Staubli VAL3: io_System.dtx

public num nLiAuto
public num nLiAux1
public num nLiAux2
public num nLiAux3
public num nLiDoorOpen
public num nLiEnd
public num nLiHome = 1
public num nLiMouldFree
public num nLiPartMade
public num nLiRobotOff
public num nLiSafety
public num nLiStart
public num nLiStop = 1
public num nLiTotalHome = 1
public num nLiWarning
public num nStateRobot
public num nLiTowerRed
public num nLiTowerYellow
public num nLiTowerGreen
public num nPowerCountCtrl
public num nLastServiceCtr
public num nLastServiceArm
public num nServiceRemain
public string sAux1
public string sAux2
public bool bBlockedCycle
public bool bBlockedUser
public bool bBtEnd
public bool bBtHome
public bool bBtRobotOff
public bool bBtStart
public bool bBtStop
public bool bCancelHomeCycl
public bool bCycleEndCalled
public bool bCycleEndPos
public bool bEnd
public bool bF7
public bool bF8
public bool bF_End
public bool bF_Home
public bool bF_Off
public bool bF_Start
public bool bF_Stop
public bool bFirstRunAfterL = true
public bool bFlashFast
public bool bFlashSlow
public bool bForceHomeReq
public bool bForceHome_ = true
public bool bHomeRetActive
public bool bModified
public bool bMouldArmInPLC
public bool bPartMade
public bool bRobotHome = true
public bool bRobotOff
public bool bRobotOffCalled
public bool bRobotOffPos
public bool bRobotZero
public bool bStartHomeCycle
public bool bStartProdCycle
public bool bTotalHome = true
public bool bUsrError
public bool btAux1
public bool btAux2
public bool btAux3
public bool bUsrWarningLow
public bool canStart
public bool canStop
public bool canResume
public bool canHom
public bool canRobotOff
public bool bRecordForce
public bool bErrorAck
public bool bUsrWarningHigh
public bool bIsEmulator
public bool bCancelEndCycle
public bool bStartInEndCycl
public jointRx jEnvMax = {j1=88.269052, j2=85.051261, j3=143.532119, j4=182.33531, j5=117.927529, j6=254.739889}
public jointRx jEnvMin = {j1=-180, j2=-47.382245, j3=-142.046726, j4=-131.97883, j5=-69.877872, j6=-189.153148}
public jointRx jPosErrCurrent = {j1=5.7E-05, j4=6.1E-05}
public jointRx jTorqueCurrent
public aio aiGrip[9]
public dio diArm[9]
public dio diBtAux1
public dio diBtAux2
public dio diBtAux3
public dio diBtEnd
public dio diBtHome
public dio diBtRobotOff
public dio diBtStart
public dio diBtStop
public dio diBtTotalHome
public dio diCore1Pos1
public dio diCore1Pos2
public dio diCore2Pos1
public dio diCore2Pos2
public dio diEjcIn
public dio diEjcOut
public dio diGrip[9]
public dio diGrip2[9]
public dio diLifeBit[2]
public dio diMachineInAuto
public dio diMouldClosed
public dio diMouldFreeFBK
public dio diMouldMidOpen
public dio diMouldOpen
public dio diRejectPart
public dio diSecuFBK[2]
public dio doAir[9]
public dio doArm[9]
public dio doAux1
public dio doAux2
public dio doCore1Pos1
public dio doCore1Pos2
public dio doCore2Pos1
public dio doCore2Pos2
public dio doEjcIn
public dio doEjcOut
public dio doFullOpening
public dio doGrip[9]
public dio doLiAuto
public dio doLiAux1
public dio doLiAux2
public dio doLiAux3
public dio doLiEnd
public dio doLiHome
public dio doLiRobotOff
public dio doLiSafety
public dio doLiStart
public dio doLiStop
public dio doLiTotalHome
public dio doMouldFree
public dio doRobotOff
public dio doSecu[2]
public dio doStartMachine
public dio doLiTowerGreen
public dio doLiTowerYellow
public dio doLiTowerRed
public dio doLiAreaFree
public dio diFuseOK[6]
public dio diSafetyPLC_OK
public dio doSignalHorn
public dio diAC_OK
public dio diLifebitsys = {link=ModbusSrv-0\Plastics-Bit\LifeBitSys}
public dio diUnusedsys = {link=ModbusSrv-0\Plastics-Bit\UnusedSys}
public dio diLifebituser = {link=ModbusSrv-0\Plastics-Bit\LifeBitUser}
public dio diUnuseduser = {link=ModbusSrv-0\Plastics-Bit\UnusedUser}
public dio diSharedbitin[32]
  [0] = {link=ModbusSrv-0\Plastics-Bit\sharedBitIn:32[0]}
  [1] = {link=ModbusSrv-0\Plastics-Bit\sharedBitIn:32[1]}
  [2] = {link=ModbusSrv-0\Plastics-Bit\sharedBitIn:32[2]}
  [3] = {link=ModbusSrv-0\Plastics-Bit\sharedBitIn:32[3]}
  [4] = {link=ModbusSrv-0\Plastics-Bit\sharedBitIn:32[4]}
  [5] = {link=ModbusSrv-0\Plastics-Bit\sharedBitIn:32[5]}
  [6] = {link=ModbusSrv-0\Plastics-Bit\sharedBitIn:32[6]}
  [7] = {link=ModbusSrv-0\Plastics-Bit\sharedBitIn:32[7]}
  [8] = {link=ModbusSrv-0\Plastics-Bit\sharedBitIn:32[8]}
  [9] = {link=ModbusSrv-0\Plastics-Bit\sharedBitIn:32[9]}
  [10] = {link=ModbusSrv-0\Plastics-Bit\sharedBitIn:32[10]}
  [11] = {link=ModbusSrv-0\Plastics-Bit\sharedBitIn:32[11]}
  [12] = {link=ModbusSrv-0\Plastics-Bit\sharedBitIn:32[12]}
  [13] = {link=ModbusSrv-0\Plastics-Bit\sharedBitIn:32[13]}
  [14] = {link=ModbusSrv-0\Plastics-Bit\sharedBitIn:32[14]}
  [15] = {link=ModbusSrv-0\Plastics-Bit\sharedBitIn:32[15]}
  [16] = {link=ModbusSrv-0\Plastics-Bit\sharedBitIn:32[16]}
  [17] = {link=ModbusSrv-0\Plastics-Bit\sharedBitIn:32[17]}
  [18] = {link=ModbusSrv-0\Plastics-Bit\sharedBitIn:32[18]}
  [19] = {link=ModbusSrv-0\Plastics-Bit\sharedBitIn:32[19]}
  [20] = {link=ModbusSrv-0\Plastics-Bit\sharedBitIn:32[20]}
  [21] = {link=ModbusSrv-0\Plastics-Bit\sharedBitIn:32[21]}
  [22] = {link=ModbusSrv-0\Plastics-Bit\sharedBitIn:32[22]}
  [23] = {link=ModbusSrv-0\Plastics-Bit\sharedBitIn:32[23]}
  [24] = {link=ModbusSrv-0\Plastics-Bit\sharedBitIn:32[24]}
  [25] = {link=ModbusSrv-0\Plastics-Bit\sharedBitIn:32[25]}
  [26] = {link=ModbusSrv-0\Plastics-Bit\sharedBitIn:32[26]}
  [27] = {link=ModbusSrv-0\Plastics-Bit\sharedBitIn:32[27]}
  [28] = {link=ModbusSrv-0\Plastics-Bit\sharedBitIn:32[28]}
  [29] = {link=ModbusSrv-0\Plastics-Bit\sharedBitIn:32[29]}
  [30] = {link=ModbusSrv-0\Plastics-Bit\sharedBitIn:32[30]}
  [31] = {link=ModbusSrv-0\Plastics-Bit\sharedBitIn:32[31]}
public dio diReserved1[63]
  [0] = {link=ModbusSrv-0\Plastics-Bit\reserved1:63[0]}
  [1] = {link=ModbusSrv-0\Plastics-Bit\reserved1:63[1]}
  [2] = {link=ModbusSrv-0\Plastics-Bit\reserved1:63[2]}
  [3] = {link=ModbusSrv-0\Plastics-Bit\reserved1:63[3]}
  [4] = {link=ModbusSrv-0\Plastics-Bit\reserved1:63[4]}
  [5] = {link=ModbusSrv-0\Plastics-Bit\reserved1:63[5]}
  [6] = {link=ModbusSrv-0\Plastics-Bit\reserved1:63[6]}
  [7] = {link=ModbusSrv-0\Plastics-Bit\reserved1:63[7]}
  [8] = {link=ModbusSrv-0\Plastics-Bit\reserved1:63[8]}
  [9] = {link=ModbusSrv-0\Plastics-Bit\reserved1:63[9]}
  [10] = {link=ModbusSrv-0\Plastics-Bit\reserved1:63[10]}
  [11] = {link=ModbusSrv-0\Plastics-Bit\reserved1:63[11]}
  [12] = {link=ModbusSrv-0\Plastics-Bit\reserved1:63[12]}
  [13] = {link=ModbusSrv-0\Plastics-Bit\reserved1:63[13]}
  [14] = {link=ModbusSrv-0\Plastics-Bit\reserved1:63[14]}
  [15] = {link=ModbusSrv-0\Plastics-Bit\reserved1:63[15]}
  [16] = {link=ModbusSrv-0\Plastics-Bit\reserved1:63[16]}
  [17] = {link=ModbusSrv-0\Plastics-Bit\reserved1:63[17]}
  [18] = {link=ModbusSrv-0\Plastics-Bit\reserved1:63[18]}
  [19] = {link=ModbusSrv-0\Plastics-Bit\reserved1:63[19]}
  [20] = {link=ModbusSrv-0\Plastics-Bit\reserved1:63[20]}
  [21] = {link=ModbusSrv-0\Plastics-Bit\reserved1:63[21]}
  [22] = {link=ModbusSrv-0\Plastics-Bit\reserved1:63[22]}
  [23] = {link=ModbusSrv-0\Plastics-Bit\reserved1:63[23]}
  [24] = {link=ModbusSrv-0\Plastics-Bit\reserved1:63[24]}
  [25] = {link=ModbusSrv-0\Plastics-Bit\reserved1:63[25]}
  [26] = {link=ModbusSrv-0\Plastics-Bit\reserved1:63[26]}
  [27] = {link=ModbusSrv-0\Plastics-Bit\reserved1:63[27]}
  [28] = {link=ModbusSrv-0\Plastics-Bit\reserved1:63[28]}
  [29] = {link=ModbusSrv-0\Plastics-Bit\reserved1:63[29]}
  [30] = {link=ModbusSrv-0\Plastics-Bit\reserved1:63[30]}
  [31] = {link=ModbusSrv-0\Plastics-Bit\reserved1:63[31]}
  [32] = {link=ModbusSrv-0\Plastics-Bit\reserved1:63[32]}
  [33] = {link=ModbusSrv-0\Plastics-Bit\reserved1:63[33]}
  [34] = {link=ModbusSrv-0\Plastics-Bit\reserved1:63[34]}
  [35] = {link=ModbusSrv-0\Plastics-Bit\reserved1:63[35]}
  [36] = {link=ModbusSrv-0\Plastics-Bit\reserved1:63[36]}
  [37] = {link=ModbusSrv-0\Plastics-Bit\reserved1:63[37]}
  [38] = {link=ModbusSrv-0\Plastics-Bit\reserved1:63[38]}
  [39] = {link=ModbusSrv-0\Plastics-Bit\reserved1:63[39]}
  [40] = {link=ModbusSrv-0\Plastics-Bit\reserved1:63[40]}
  [41] = {link=ModbusSrv-0\Plastics-Bit\reserved1:63[41]}
  [42] = {link=ModbusSrv-0\Plastics-Bit\reserved1:63[42]}
  [43] = {link=ModbusSrv-0\Plastics-Bit\reserved1:63[43]}
  [44] = {link=ModbusSrv-0\Plastics-Bit\reserved1:63[44]}
  [45] = {link=ModbusSrv-0\Plastics-Bit\reserved1:63[45]}
  [46] = {link=ModbusSrv-0\Plastics-Bit\reserved1:63[46]}
  [47] = {link=ModbusSrv-0\Plastics-Bit\reserved1:63[47]}
  [48] = {link=ModbusSrv-0\Plastics-Bit\reserved1:63[48]}
  [49] = {link=ModbusSrv-0\Plastics-Bit\reserved1:63[49]}
  [50] = {link=ModbusSrv-0\Plastics-Bit\reserved1:63[50]}
  [51] = {link=ModbusSrv-0\Plastics-Bit\reserved1:63[51]}
  [52] = {link=ModbusSrv-0\Plastics-Bit\reserved1:63[52]}
  [53] = {link=ModbusSrv-0\Plastics-Bit\reserved1:63[53]}
  [54] = {link=ModbusSrv-0\Plastics-Bit\reserved1:63[54]}
  [55] = {link=ModbusSrv-0\Plastics-Bit\reserved1:63[55]}
  [56] = {link=ModbusSrv-0\Plastics-Bit\reserved1:63[56]}
  [57] = {link=ModbusSrv-0\Plastics-Bit\reserved1:63[57]}
  [58] = {link=ModbusSrv-0\Plastics-Bit\reserved1:63[58]}
  [59] = {link=ModbusSrv-0\Plastics-Bit\reserved1:63[59]}
  [60] = {link=ModbusSrv-0\Plastics-Bit\reserved1:63[60]}
  [61] = {link=ModbusSrv-0\Plastics-Bit\reserved1:63[61]}
  [62] = {link=ModbusSrv-0\Plastics-Bit\reserved1:63[62]}
public dio doN1_102[8]
  [0] = {link=ModbusSrv-0\Plastics-Bit\N1_102:8[0]}
  [1] = {link=ModbusSrv-0\Plastics-Bit\N1_102:8[1]}
  [2] = {link=ModbusSrv-0\Plastics-Bit\N1_102:8[2]}
  [3] = {link=ModbusSrv-0\Plastics-Bit\N1_102:8[3]}
  [4] = {link=ModbusSrv-0\Plastics-Bit\N1_102:8[4]}
  [5] = {link=ModbusSrv-0\Plastics-Bit\N1_102:8[5]}
  [6] = {link=ModbusSrv-0\Plastics-Bit\N1_102:8[6]}
  [7] = {link=ModbusSrv-0\Plastics-Bit\N1_102:8[7]}
public dio doN1_103[8]
  [0] = {link=ModbusSrv-0\Plastics-Bit\N1_103:8[0]}
  [1] = {link=ModbusSrv-0\Plastics-Bit\N1_103:8[1]}
  [2] = {link=ModbusSrv-0\Plastics-Bit\N1_103:8[2]}
  [3] = {link=ModbusSrv-0\Plastics-Bit\N1_103:8[3]}
  [4] = {link=ModbusSrv-0\Plastics-Bit\N1_103:8[4]}
  [5] = {link=ModbusSrv-0\Plastics-Bit\N1_103:8[5]}
  [6] = {link=ModbusSrv-0\Plastics-Bit\N1_103:8[6]}
  [7] = {link=ModbusSrv-0\Plastics-Bit\N1_103:8[7]}
public dio doN1_202[8]
  [0] = {link=ModbusSrv-0\Plastics-Bit\N1_202:8[0]}
  [1] = {link=ModbusSrv-0\Plastics-Bit\N1_202:8[1]}
  [2] = {link=ModbusSrv-0\Plastics-Bit\N1_202:8[2]}
  [3] = {link=ModbusSrv-0\Plastics-Bit\N1_202:8[3]}
  [4] = {link=ModbusSrv-0\Plastics-Bit\N1_202:8[4]}
  [5] = {link=ModbusSrv-0\Plastics-Bit\N1_202:8[5]}
  [6] = {link=ModbusSrv-0\Plastics-Bit\N1_202:8[6]}
  [7] = {link=ModbusSrv-0\Plastics-Bit\N1_202:8[7]}
public dio doN1_303[4]
  [0] = {link=ModbusSrv-0\Plastics-Bit\N1_303:4[0]}
  [1] = {link=ModbusSrv-0\Plastics-Bit\N1_303:4[1]}
  [2] = {link=ModbusSrv-0\Plastics-Bit\N1_303:4[2]}
  [3] = {link=ModbusSrv-0\Plastics-Bit\N1_303:4[3]}
public dio doN1_305[2]
  [0] = {link=ModbusSrv-0\Plastics-Bit\N1_305:2[0]}
  [1] = {link=ModbusSrv-0\Plastics-Bit\N1_305:2[1]}
public dio doN1_306[2]
  [0] = {link=ModbusSrv-0\Plastics-Bit\N1_306:2[0]}
  [1] = {link=ModbusSrv-0\Plastics-Bit\N1_306:2[1]}
public dio doN1_307[2]
  [0] = {link=ModbusSrv-0\Plastics-Bit\N1_307:2[0]}
  [1] = {link=ModbusSrv-0\Plastics-Bit\N1_307:2[1]}
public dio doN1_308[2]
  [0] = {link=ModbusSrv-0\Plastics-Bit\N1_308:2[0]}
  [1] = {link=ModbusSrv-0\Plastics-Bit\N1_308:2[1]}
public dio doN1_309[2]
  [0] = {link=ModbusSrv-0\Plastics-Bit\N1_309:2[0]}
  [1] = {link=ModbusSrv-0\Plastics-Bit\N1_309:2[1]}
public dio doN2_104[8]
  [0] = {link=ModbusSrv-0\Plastics-Bit\N2_104:8[0]}
  [1] = {link=ModbusSrv-0\Plastics-Bit\N2_104:8[1]}
  [2] = {link=ModbusSrv-0\Plastics-Bit\N2_104:8[2]}
  [3] = {link=ModbusSrv-0\Plastics-Bit\N2_104:8[3]}
  [4] = {link=ModbusSrv-0\Plastics-Bit\N2_104:8[4]}
  [5] = {link=ModbusSrv-0\Plastics-Bit\N2_104:8[5]}
  [6] = {link=ModbusSrv-0\Plastics-Bit\N2_104:8[6]}
  [7] = {link=ModbusSrv-0\Plastics-Bit\N2_104:8[7]}
public dio doN2_105[8]
  [0] = {link=ModbusSrv-0\Plastics-Bit\N2_105:8[0]}
  [1] = {link=ModbusSrv-0\Plastics-Bit\N2_105:8[1]}
  [2] = {link=ModbusSrv-0\Plastics-Bit\N2_105:8[2]}
  [3] = {link=ModbusSrv-0\Plastics-Bit\N2_105:8[3]}
  [4] = {link=ModbusSrv-0\Plastics-Bit\N2_105:8[4]}
  [5] = {link=ModbusSrv-0\Plastics-Bit\N2_105:8[5]}
  [6] = {link=ModbusSrv-0\Plastics-Bit\N2_105:8[6]}
  [7] = {link=ModbusSrv-0\Plastics-Bit\N2_105:8[7]}
public dio doN2_106[8]
  [0] = {link=ModbusSrv-0\Plastics-Bit\N2_106:8[0]}
  [1] = {link=ModbusSrv-0\Plastics-Bit\N2_106:8[1]}
  [2] = {link=ModbusSrv-0\Plastics-Bit\N2_106:8[2]}
  [3] = {link=ModbusSrv-0\Plastics-Bit\N2_106:8[3]}
  [4] = {link=ModbusSrv-0\Plastics-Bit\N2_106:8[4]}
  [5] = {link=ModbusSrv-0\Plastics-Bit\N2_106:8[5]}
  [6] = {link=ModbusSrv-0\Plastics-Bit\N2_106:8[6]}
  [7] = {link=ModbusSrv-0\Plastics-Bit\N2_106:8[7]}
public dio doN2_107[8]
  [0] = {link=ModbusSrv-0\Plastics-Bit\N2_107:8[0]}
  [1] = {link=ModbusSrv-0\Plastics-Bit\N2_107:8[1]}
  [2] = {link=ModbusSrv-0\Plastics-Bit\N2_107:8[2]}
  [3] = {link=ModbusSrv-0\Plastics-Bit\N2_107:8[3]}
  [4] = {link=ModbusSrv-0\Plastics-Bit\N2_107:8[4]}
  [5] = {link=ModbusSrv-0\Plastics-Bit\N2_107:8[5]}
  [6] = {link=ModbusSrv-0\Plastics-Bit\N2_107:8[6]}
  [7] = {link=ModbusSrv-0\Plastics-Bit\N2_107:8[7]}
public dio doSharedbitout[32]
  [0] = {link=ModbusSrv-0\Plastics-Bit\sharedBitOut:32[0]}
  [1] = {link=ModbusSrv-0\Plastics-Bit\sharedBitOut:32[1]}
  [2] = {link=ModbusSrv-0\Plastics-Bit\sharedBitOut:32[2]}
  [3] = {link=ModbusSrv-0\Plastics-Bit\sharedBitOut:32[3]}
  [4] = {link=ModbusSrv-0\Plastics-Bit\sharedBitOut:32[4]}
  [5] = {link=ModbusSrv-0\Plastics-Bit\sharedBitOut:32[5]}
  [6] = {link=ModbusSrv-0\Plastics-Bit\sharedBitOut:32[6]}
  [7] = {link=ModbusSrv-0\Plastics-Bit\sharedBitOut:32[7]}
  [8] = {link=ModbusSrv-0\Plastics-Bit\sharedBitOut:32[8]}
  [9] = {link=ModbusSrv-0\Plastics-Bit\sharedBitOut:32[9]}
  [10] = {link=ModbusSrv-0\Plastics-Bit\sharedBitOut:32[10]}
  [11] = {link=ModbusSrv-0\Plastics-Bit\sharedBitOut:32[11]}
  [12] = {link=ModbusSrv-0\Plastics-Bit\sharedBitOut:32[12]}
  [13] = {link=ModbusSrv-0\Plastics-Bit\sharedBitOut:32[13]}
  [14] = {link=ModbusSrv-0\Plastics-Bit\sharedBitOut:32[14]}
  [15] = {link=ModbusSrv-0\Plastics-Bit\sharedBitOut:32[15]}
  [16] = {link=ModbusSrv-0\Plastics-Bit\sharedBitOut:32[16]}
  [17] = {link=ModbusSrv-0\Plastics-Bit\sharedBitOut:32[17]}
  [18] = {link=ModbusSrv-0\Plastics-Bit\sharedBitOut:32[18]}
  [19] = {link=ModbusSrv-0\Plastics-Bit\sharedBitOut:32[19]}
  [20] = {link=ModbusSrv-0\Plastics-Bit\sharedBitOut:32[20]}
  [21] = {link=ModbusSrv-0\Plastics-Bit\sharedBitOut:32[21]}
  [22] = {link=ModbusSrv-0\Plastics-Bit\sharedBitOut:32[22]}
  [23] = {link=ModbusSrv-0\Plastics-Bit\sharedBitOut:32[23]}
  [24] = {link=ModbusSrv-0\Plastics-Bit\sharedBitOut:32[24]}
  [25] = {link=ModbusSrv-0\Plastics-Bit\sharedBitOut:32[25]}
  [26] = {link=ModbusSrv-0\Plastics-Bit\sharedBitOut:32[26]}
  [27] = {link=ModbusSrv-0\Plastics-Bit\sharedBitOut:32[27]}
  [28] = {link=ModbusSrv-0\Plastics-Bit\sharedBitOut:32[28]}
  [29] = {link=ModbusSrv-0\Plastics-Bit\sharedBitOut:32[29]}
  [30] = {link=ModbusSrv-0\Plastics-Bit\sharedBitOut:32[30]}
  [31] = {link=ModbusSrv-0\Plastics-Bit\sharedBitOut:32[31]}
public dio doBrakeselect = {link=ModbusSrv-0\Plastics-Bit\brakeSelect}
public dio doDoor = {link=ModbusSrv-0\Plastics-Bit\door}
public dio doEstopes34 = {link=ModbusSrv-0\Plastics-Bit\estopES34}
public dio doEstopes12 = {link=ModbusSrv-0\Plastics-Bit\estopES12}
public dio doEstopmcp = {link=ModbusSrv-0\Plastics-Bit\estopMCP}
public dio doLimitswitch = {link=ModbusSrv-0\Plastics-Bit\limitSwitch}
public dio doDdummy[8]
  [0] = {link=ModbusSrv-0\Plastics-Bit\dDummy:8[0]}
  [1] = {link=ModbusSrv-0\Plastics-Bit\dDummy:8[1]}
  [2] = {link=ModbusSrv-0\Plastics-Bit\dDummy:8[2]}
  [3] = {link=ModbusSrv-0\Plastics-Bit\dDummy:8[3]}
  [4] = {link=ModbusSrv-0\Plastics-Bit\dDummy:8[4]}
  [5] = {link=ModbusSrv-0\Plastics-Bit\dDummy:8[5]}
  [6] = {link=ModbusSrv-0\Plastics-Bit\dDummy:8[6]}
  [7] = {link=ModbusSrv-0\Plastics-Bit\dDummy:8[7]}
public dio doPower = {link=ModbusSrv-0\Plastics-Bit\power}
public dio doByte0[8]
  [0] = {link=ModbusSrv-0\Plastics-Bit\byte0:8[0]}
  [1] = {link=ModbusSrv-0\Plastics-Bit\byte0:8[1]}
  [2] = {link=ModbusSrv-0\Plastics-Bit\byte0:8[2]}
  [3] = {link=ModbusSrv-0\Plastics-Bit\byte0:8[3]}
  [4] = {link=ModbusSrv-0\Plastics-Bit\byte0:8[4]}
  [5] = {link=ModbusSrv-0\Plastics-Bit\byte0:8[5]}
  [6] = {link=ModbusSrv-0\Plastics-Bit\byte0:8[6]}
  [7] = {link=ModbusSrv-0\Plastics-Bit\byte0:8[7]}
public dio doByte1[8]
  [0] = {link=ModbusSrv-0\Plastics-Bit\byte1:8[0]}
  [1] = {link=ModbusSrv-0\Plastics-Bit\byte1:8[1]}
  [2] = {link=ModbusSrv-0\Plastics-Bit\byte1:8[2]}
  [3] = {link=ModbusSrv-0\Plastics-Bit\byte1:8[3]}
  [4] = {link=ModbusSrv-0\Plastics-Bit\byte1:8[4]}
  [5] = {link=ModbusSrv-0\Plastics-Bit\byte1:8[5]}
  [6] = {link=ModbusSrv-0\Plastics-Bit\byte1:8[6]}
  [7] = {link=ModbusSrv-0\Plastics-Bit\byte1:8[7]}
public dio doByte2[8]
  [0] = {link=ModbusSrv-0\Plastics-Bit\byte2:8[0]}
  [1] = {link=ModbusSrv-0\Plastics-Bit\byte2:8[1]}
  [2] = {link=ModbusSrv-0\Plastics-Bit\byte2:8[2]}
  [3] = {link=ModbusSrv-0\Plastics-Bit\byte2:8[3]}
  [4] = {link=ModbusSrv-0\Plastics-Bit\byte2:8[4]}
  [5] = {link=ModbusSrv-0\Plastics-Bit\byte2:8[5]}
  [6] = {link=ModbusSrv-0\Plastics-Bit\byte2:8[6]}
  [7] = {link=ModbusSrv-0\Plastics-Bit\byte2:8[7]}
public dio doByte3[8]
  [0] = {link=ModbusSrv-0\Plastics-Bit\byte3:8[0]}
  [1] = {link=ModbusSrv-0\Plastics-Bit\byte3:8[1]}
  [2] = {link=ModbusSrv-0\Plastics-Bit\byte3:8[2]}
  [3] = {link=ModbusSrv-0\Plastics-Bit\byte3:8[3]}
  [4] = {link=ModbusSrv-0\Plastics-Bit\byte3:8[4]}
  [5] = {link=ModbusSrv-0\Plastics-Bit\byte3:8[5]}
  [6] = {link=ModbusSrv-0\Plastics-Bit\byte3:8[6]}
  [7] = {link=ModbusSrv-0\Plastics-Bit\byte3:8[7]}
public dio doAgripper[16]
  [0] = {link=ModbusSrv-0\Plastics-Bit\aGripper:16[0]}
  [1] = {link=ModbusSrv-0\Plastics-Bit\aGripper:16[1]}
  [2] = {link=ModbusSrv-0\Plastics-Bit\aGripper:16[2]}
  [3] = {link=ModbusSrv-0\Plastics-Bit\aGripper:16[3]}
  [4] = {link=ModbusSrv-0\Plastics-Bit\aGripper:16[4]}
  [5] = {link=ModbusSrv-0\Plastics-Bit\aGripper:16[5]}
  [6] = {link=ModbusSrv-0\Plastics-Bit\aGripper:16[6]}
  [7] = {link=ModbusSrv-0\Plastics-Bit\aGripper:16[7]}
  [8] = {link=ModbusSrv-0\Plastics-Bit\aGripper:16[8]}
  [9] = {link=ModbusSrv-0\Plastics-Bit\aGripper:16[9]}
  [10] = {link=ModbusSrv-0\Plastics-Bit\aGripper:16[10]}
  [11] = {link=ModbusSrv-0\Plastics-Bit\aGripper:16[11]}
  [12] = {link=ModbusSrv-0\Plastics-Bit\aGripper:16[12]}
  [13] = {link=ModbusSrv-0\Plastics-Bit\aGripper:16[13]}
  [14] = {link=ModbusSrv-0\Plastics-Bit\aGripper:16[14]}
  [15] = {link=ModbusSrv-0\Plastics-Bit\aGripper:16[15]}
public aio aiDummyword[2]
  [0] = {link=ModbusSrv-0\Plastics-Word\dummyWord:2[0]}
  [1] = {link=ModbusSrv-0\Plastics-Word\dummyWord:2[1]}
public aio aiN1_200[4]
  [0] = {link=ModbusSrv-0\Plastics-Word\N1_200:4[0]}
  [1] = {link=ModbusSrv-0\Plastics-Word\N1_200:4[1]}
  [2] = {link=ModbusSrv-0\Plastics-Word\N1_200:4[2]}
  [3] = {link=ModbusSrv-0\Plastics-Word\N1_200:4[3]}
public aio aiSharedwordin[16]
  [0] = {link=ModbusSrv-0\Plastics-Word\sharedWordIn:16[0]}
  [1] = {link=ModbusSrv-0\Plastics-Word\sharedWordIn:16[1]}
  [2] = {link=ModbusSrv-0\Plastics-Word\sharedWordIn:16[2]}
  [3] = {link=ModbusSrv-0\Plastics-Word\sharedWordIn:16[3]}
  [4] = {link=ModbusSrv-0\Plastics-Word\sharedWordIn:16[4]}
  [5] = {link=ModbusSrv-0\Plastics-Word\sharedWordIn:16[5]}
  [6] = {link=ModbusSrv-0\Plastics-Word\sharedWordIn:16[6]}
  [7] = {link=ModbusSrv-0\Plastics-Word\sharedWordIn:16[7]}
  [8] = {link=ModbusSrv-0\Plastics-Word\sharedWordIn:16[8]}
  [9] = {link=ModbusSrv-0\Plastics-Word\sharedWordIn:16[9]}
  [10] = {link=ModbusSrv-0\Plastics-Word\sharedWordIn:16[10]}
  [11] = {link=ModbusSrv-0\Plastics-Word\sharedWordIn:16[11]}
  [12] = {link=ModbusSrv-0\Plastics-Word\sharedWordIn:16[12]}
  [13] = {link=ModbusSrv-0\Plastics-Word\sharedWordIn:16[13]}
  [14] = {link=ModbusSrv-0\Plastics-Word\sharedWordIn:16[14]}
  [15] = {link=ModbusSrv-0\Plastics-Word\sharedWordIn:16[15]}
public aio aiSharedwordout[16]
  [0] = {link=ModbusSrv-0\Plastics-Word\sharedWordOut:16[0]}
  [1] = {link=ModbusSrv-0\Plastics-Word\sharedWordOut:16[1]}
  [2] = {link=ModbusSrv-0\Plastics-Word\sharedWordOut:16[2]}
  [3] = {link=ModbusSrv-0\Plastics-Word\sharedWordOut:16[3]}
  [4] = {link=ModbusSrv-0\Plastics-Word\sharedWordOut:16[4]}
  [5] = {link=ModbusSrv-0\Plastics-Word\sharedWordOut:16[5]}
  [6] = {link=ModbusSrv-0\Plastics-Word\sharedWordOut:16[6]}
  [7] = {link=ModbusSrv-0\Plastics-Word\sharedWordOut:16[7]}
  [8] = {link=ModbusSrv-0\Plastics-Word\sharedWordOut:16[8]}
  [9] = {link=ModbusSrv-0\Plastics-Word\sharedWordOut:16[9]}
  [10] = {link=ModbusSrv-0\Plastics-Word\sharedWordOut:16[10]}
  [11] = {link=ModbusSrv-0\Plastics-Word\sharedWordOut:16[11]}
  [12] = {link=ModbusSrv-0\Plastics-Word\sharedWordOut:16[12]}
  [13] = {link=ModbusSrv-0\Plastics-Word\sharedWordOut:16[13]}
  [14] = {link=ModbusSrv-0\Plastics-Word\sharedWordOut:16[14]}
  [15] = {link=ModbusSrv-0\Plastics-Word\sharedWordOut:16[15]}
public dio N1_100[8] = {link=ModbusSrv-0\Plastics-Bit\N1_100:8[0]}
